KUKA KRL program: ServiceTmpReadMe.src

&ACCESS RVP
&COMMENT ReadMe File
DEF  ServiceTmpReadMe ( )

; This file only exists as a directory placeholder file.

END
